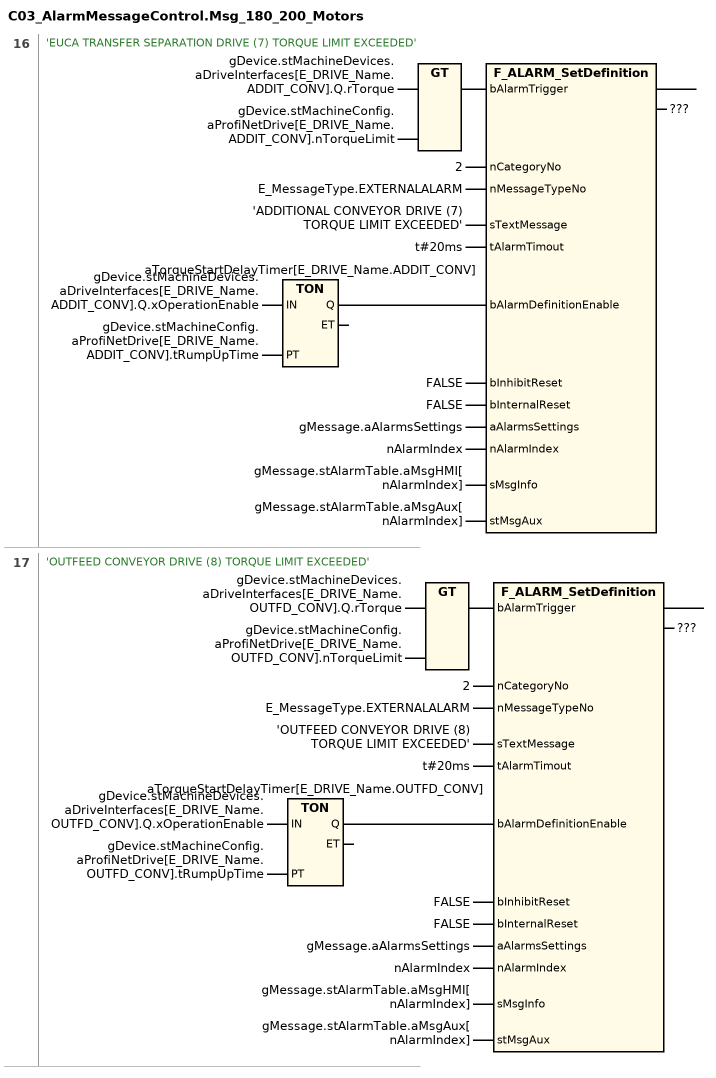
// NETWORK 16
// 'EUCA TRANSFER SEPARATION DRIVE (7) TORQUE LIMIT EXCEEDED'
aTorqueStartDelayTimer[E_DRIVE_Name.ADDIT_CONV](IN := gDevice.stMachineDevices.aDriveInterfaces[E_DRIVE_Name.ADDIT_CONV].Q.xOperationEnable, PT := gDevice.stMachineConfig.aProfiNetDrive[E_DRIVE_Name.ADDIT_CONV].tRumpUpTime); // TON
F_ALARM_SetDefinition(bAlarmTrigger := gDevice.stMachineDevices.aDriveInterfaces[E_DRIVE_Name.ADDIT_CONV].Q.rTorque > gDevice.stMachineConfig.aProfiNetDrive[E_DRIVE_Name.ADDIT_CONV].nTorqueLimit, nCategoryNo := 2, nMessageTypeNo := E_MessageType.EXTERNALALARM, sTextMessage := 'ADDITIONAL CONVEYOR DRIVE (7) TORQUE LIMIT EXCEEDED', tAlarmTimout := t#20ms, bAlarmDefinitionEnable := aTorqueStartDelayTimer[E_DRIVE_Name.ADDIT_CONV].Q, bInhibitReset := FALSE, bInternalReset := FALSE, aAlarmsSettings := gMessage.aAlarmsSettings, nAlarmIndex := nAlarmIndex, sMsgInfo := gMessage.stAlarmTable.aMsgHMI[nAlarmIndex], stMsgAux := gMessage.stAlarmTable.aMsgAux[nAlarmIndex]);

// NETWORK 17
// 'OUTFEED CONVEYOR DRIVE (8) TORQUE LIMIT EXCEEDED'
aTorqueStartDelayTimer[E_DRIVE_Name.OUTFD_CONV](IN := gDevice.stMachineDevices.aDriveInterfaces[E_DRIVE_Name.OUTFD_CONV].Q.xOperationEnable, PT := gDevice.stMachineConfig.aProfiNetDrive[E_DRIVE_Name.OUTFD_CONV].tRumpUpTime); // TON
F_ALARM_SetDefinition(bAlarmTrigger := gDevice.stMachineDevices.aDriveInterfaces[E_DRIVE_Name.OUTFD_CONV].Q.rTorque > gDevice.stMachineConfig.aProfiNetDrive[E_DRIVE_Name.OUTFD_CONV].nTorqueLimit, nCategoryNo := 2, nMessageTypeNo := E_MessageType.EXTERNALALARM, sTextMessage := 'OUTFEED CONVEYOR DRIVE (8) TORQUE LIMIT EXCEEDED', tAlarmTimout := t#20ms, bAlarmDefinitionEnable := aTorqueStartDelayTimer[E_DRIVE_Name.OUTFD_CONV].Q, bInhibitReset := FALSE, bInternalReset := FALSE, aAlarmsSettings := gMessage.aAlarmsSettings, nAlarmIndex := nAlarmIndex, sMsgInfo := gMessage.stAlarmTable.aMsgHMI[nAlarmIndex], stMsgAux := gMessage.stAlarmTable.aMsgAux[nAlarmIndex]);

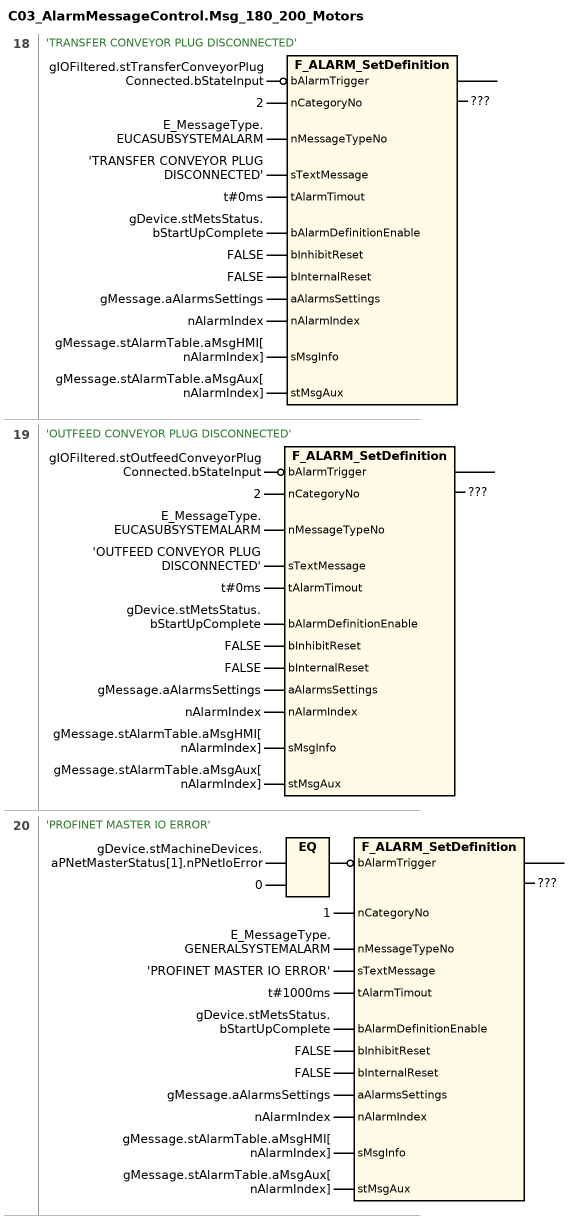
// NETWORK 18
// 'TRANSFER CONVEYOR PLUG DISCONNECTED'
F_ALARM_SetDefinition(bAlarmTrigger := NOT gIOFiltered.stTransferConveyorPlugConnected.bStateInput, nCategoryNo := 2, nMessageTypeNo := E_MessageType.EUCASUBSYSTEMALARM, sTextMessage := 'TRANSFER CONVEYOR PLUG DISCONNECTED', tAlarmTimout := t#0ms, bAlarmDefinitionEnable := gDevice.stMetsStatus.bStartUpComplete, bInhibitReset := FALSE, bInternalReset := FALSE, aAlarmsSettings := gMessage.aAlarmsSettings, nAlarmIndex := nAlarmIndex, sMsgInfo := gMessage.stAlarmTable.aMsgHMI[nAlarmIndex], stMsgAux := gMessage.stAlarmTable.aMsgAux[nAlarmIndex]);

// NETWORK 19
// 'OUTFEED CONVEYOR PLUG DISCONNECTED'
F_ALARM_SetDefinition(bAlarmTrigger := NOT gIOFiltered.stOutfeedConveyorPlugConnected.bStateInput, nCategoryNo := 2, nMessageTypeNo := E_MessageType.EUCASUBSYSTEMALARM, sTextMessage := 'OUTFEED CONVEYOR PLUG DISCONNECTED', tAlarmTimout := t#0ms, bAlarmDefinitionEnable := gDevice.stMetsStatus.bStartUpComplete, bInhibitReset := FALSE, bInternalReset := FALSE, aAlarmsSettings := gMessage.aAlarmsSettings, nAlarmIndex := nAlarmIndex, sMsgInfo := gMessage.stAlarmTable.aMsgHMI[nAlarmIndex], stMsgAux := gMessage.stAlarmTable.aMsgAux[nAlarmIndex]);

// NETWORK 20
// 'PROFINET MASTER IO ERROR'
F_ALARM_SetDefinition(bAlarmTrigger := NOT (gDevice.stMachineDevices.aPNetMasterStatus[1].nPNetIoError = 0), nCategoryNo := 1, nMessageTypeNo := E_MessageType.GENERALSYSTEMALARM, sTextMessage := 'PROFINET MASTER IO ERROR', tAlarmTimout := t#1000ms, bAlarmDefinitionEnable := gDevice.stMetsStatus.bStartUpComplete, bInhibitReset := FALSE, bInternalReset := FALSE, aAlarmsSettings := gMessage.aAlarmsSettings, nAlarmIndex := nAlarmIndex, sMsgInfo := gMessage.stAlarmTable.aMsgHMI[nAlarmIndex], stMsgAux := gMessage.stAlarmTable.aMsgAux[nAlarmIndex]);

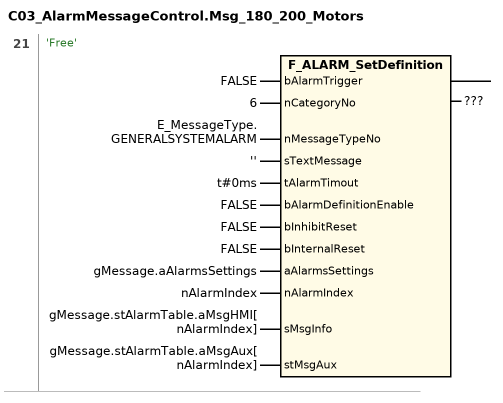
// NETWORK 21
// 'Free'
F_ALARM_SetDefinition(bAlarmTrigger := FALSE, nCategoryNo := 6, nMessageTypeNo := E_MessageType.GENERALSYSTEMALARM, sTextMessage := '', tAlarmTimout := t#0ms, bAlarmDefinitionEnable := FALSE, bInhibitReset := FALSE, bInternalReset := FALSE, aAlarmsSettings := gMessage.aAlarmsSettings, nAlarmIndex := nAlarmIndex, sMsgInfo := gMessage.stAlarmTable.aMsgHMI[nAlarmIndex], stMsgAux := gMessage.stAlarmTable.aMsgAux[nAlarmIndex]);
END_ACTION

ACTION Msg_201_208_Interface:
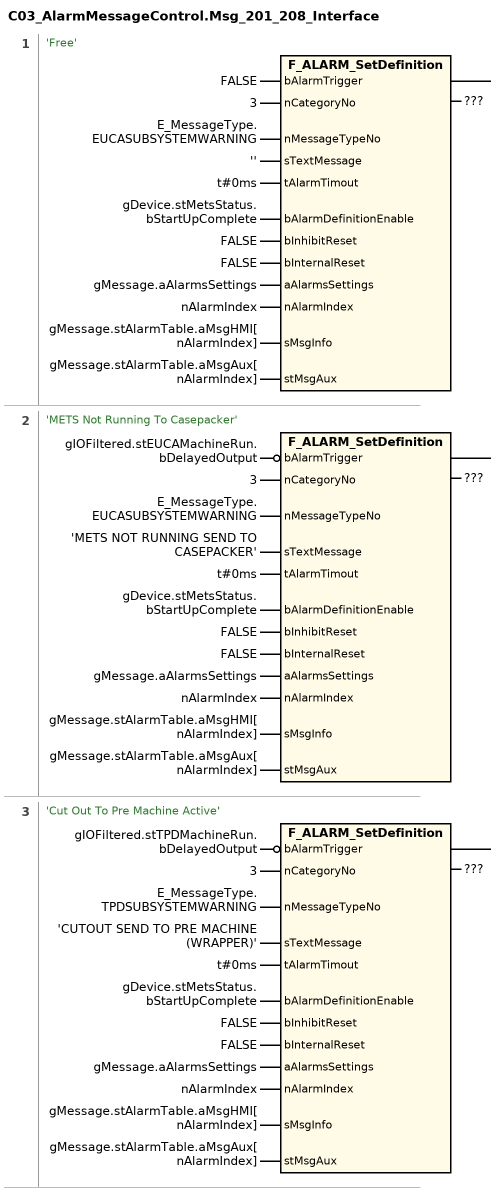
// NETWORK 1
// 'Free'
F_ALARM_SetDefinition(bAlarmTrigger := FALSE, nCategoryNo := 3, nMessageTypeNo := E_MessageType.EUCASUBSYSTEMWARNING, sTextMessage := '', tAlarmTimout := t#0ms, bAlarmDefinitionEnable := gDevice.stMetsStatus.bStartUpComplete, bInhibitReset := FALSE, bInternalReset := FALSE, aAlarmsSettings := gMessage.aAlarmsSettings, nAlarmIndex := nAlarmIndex, sMsgInfo := gMessage.stAlarmTable.aMsgHMI[nAlarmIndex], stMsgAux := gMessage.stAlarmTable.aMsgAux[nAlarmIndex]);

// NETWORK 2
// 'METS Not Running To Casepacker'
F_ALARM_SetDefinition(bAlarmTrigger := NOT gIOFiltered.stEUCAMachineRun.bDelayedOutput, nCategoryNo := 3, nMessageTypeNo := E_MessageType.EUCASUBSYSTEMWARNING, sTextMessage := 'METS NOT RUNNING SEND TO CASEPACKER', tAlarmTimout := t#0ms, bAlarmDefinitionEnable := gDevice.stMetsStatus.bStartUpComplete, bInhibitReset := FALSE, bInternalReset := FALSE, aAlarmsSettings := gMessage.aAlarmsSettings, nAlarmIndex := nAlarmIndex, sMsgInfo := gMessage.stAlarmTable.aMsgHMI[nAlarmIndex], stMsgAux := gMessage.stAlarmTable.aMsgAux[nAlarmIndex]);

// NETWORK 3
// 'Cut Out To Pre Machine Active'
F_ALARM_SetDefinition(bAlarmTrigger := NOT gIOFiltered.stTPDMachineRun.bDelayedOutput, nCategoryNo := 3, nMessageTypeNo := E_MessageType.TPDSUBSYSTEMWARNING, sTextMessage := 'CUTOUT SEND TO PRE MACHINE (WRAPPER)', tAlarmTimout := t#0ms, bAlarmDefinitionEnable := gDevice.stMetsStatus.bStartUpComplete, bInhibitReset := FALSE, bInternalReset := FALSE, aAlarmsSettings := gMessage.aAlarmsSettings, nAlarmIndex := nAlarmIndex, sMsgInfo := gMessage.stAlarmTable.aMsgHMI[nAlarmIndex], stMsgAux := gMessage.stAlarmTable.aMsgAux[nAlarmIndex]);

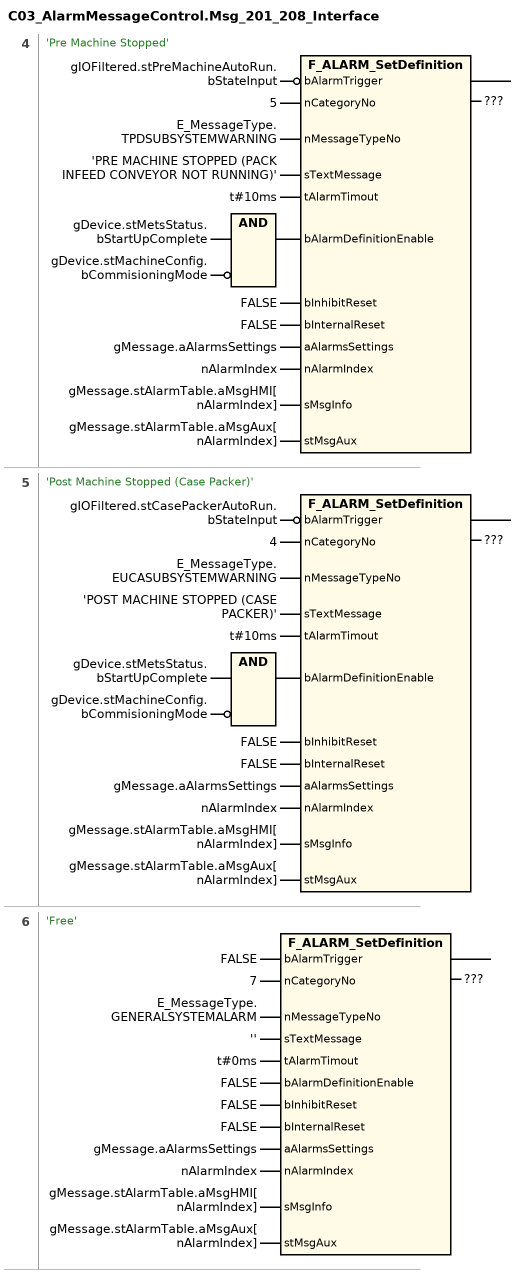
// NETWORK 4
// 'Pre Machine Stopped'
F_ALARM_SetDefinition(bAlarmTrigger := NOT gIOFiltered.stPreMachineAutoRun.bStateInput, nCategoryNo := 5, nMessageTypeNo := E_MessageType.TPDSUBSYSTEMWARNING, sTextMessage := 'PRE MACHINE STOPPED (PACK INFEED CONVEYOR NOT RUNNING)', tAlarmTimout := t#10ms, bAlarmDefinitionEnable := gDevice.stMetsStatus.bStartUpComplete AND NOT gDevice.stMachineConfig.bCommisioningMode, bInhibitReset := FALSE, bInternalReset := FALSE, aAlarmsSettings := gMessage.aAlarmsSettings, nAlarmIndex := nAlarmIndex, sMsgInfo := gMessage.stAlarmTable.aMsgHMI[nAlarmIndex], stMsgAux := gMessage.stAlarmTable.aMsgAux[nAlarmIndex]);

// NETWORK 5
// 'Post Machine Stopped (Case Packer)'
F_ALARM_SetDefinition(bAlarmTrigger := NOT gIOFiltered.stCasePackerAutoRun.bStateInput, nCategoryNo := 4, nMessageTypeNo := E_MessageType.EUCASUBSYSTEMWARNING, sTextMessage := 'POST MACHINE STOPPED (CASE PACKER)', tAlarmTimout := t#10ms, bAlarmDefinitionEnable := gDevice.stMetsStatus.bStartUpComplete AND NOT gDevice.stMachineConfig.bCommisioningMode, bInhibitReset := FALSE, bInternalReset := FALSE, aAlarmsSettings := gMessage.aAlarmsSettings, nAlarmIndex := nAlarmIndex, sMsgInfo := gMessage.stAlarmTable.aMsgHMI[nAlarmIndex], stMsgAux := gMessage.stAlarmTable.aMsgAux[nAlarmIndex]);

// NETWORK 6
// 'Free'
F_ALARM_SetDefinition(bAlarmTrigger := FALSE, nCategoryNo := 7, nMessageTypeNo := E_MessageType.GENERALSYSTEMALARM, sTextMessage := '', tAlarmTimout := t#0ms, bAlarmDefinitionEnable := FALSE, bInhibitReset := FALSE, bInternalReset := FALSE, aAlarmsSettings := gMessage.aAlarmsSettings, nAlarmIndex := nAlarmIndex, sMsgInfo := gMessage.stAlarmTable.aMsgHMI[nAlarmIndex], stMsgAux := gMessage.stAlarmTable.aMsgAux[nAlarmIndex]);

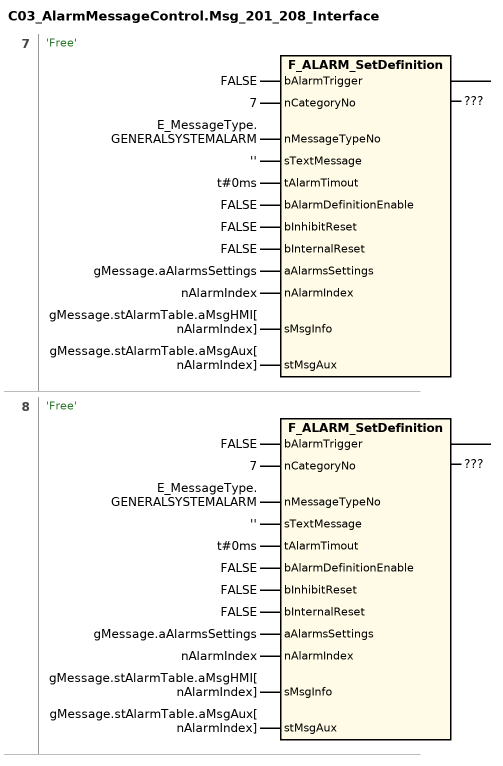
// NETWORK 7
// 'Free'
F_ALARM_SetDefinition(bAlarmTrigger := FALSE, nCategoryNo := 7, nMessageTypeNo := E_MessageType.GENERALSYSTEMALARM, sTextMessage := '', tAlarmTimout := t#0ms, bAlarmDefinitionEnable := FALSE, bInhibitReset := FALSE, bInternalReset := FALSE, aAlarmsSettings := gMessage.aAlarmsSettings, nAlarmIndex := nAlarmIndex, sMsgInfo := gMessage.stAlarmTable.aMsgHMI[nAlarmIndex], stMsgAux := gMessage.stAlarmTable.aMsgAux[nAlarmIndex]);

// NETWORK 8
// 'Free'
F_ALARM_SetDefinition(bAlarmTrigger := FALSE, nCategoryNo := 7, nMessageTypeNo := E_MessageType.GENERALSYSTEMALARM, sTextMessage := '', tAlarmTimout := t#0ms, bAlarmDefinitionEnable := FALSE, bInhibitReset := FALSE, bInternalReset := FALSE, aAlarmsSettings := gMessage.aAlarmsSettings, nAlarmIndex := nAlarmIndex, sMsgInfo := gMessage.stAlarmTable.aMsgHMI[nAlarmIndex], stMsgAux := gMessage.stAlarmTable.aMsgAux[nAlarmIndex]);
END_ACTION

ACTION Msg_209_237_Labellers:
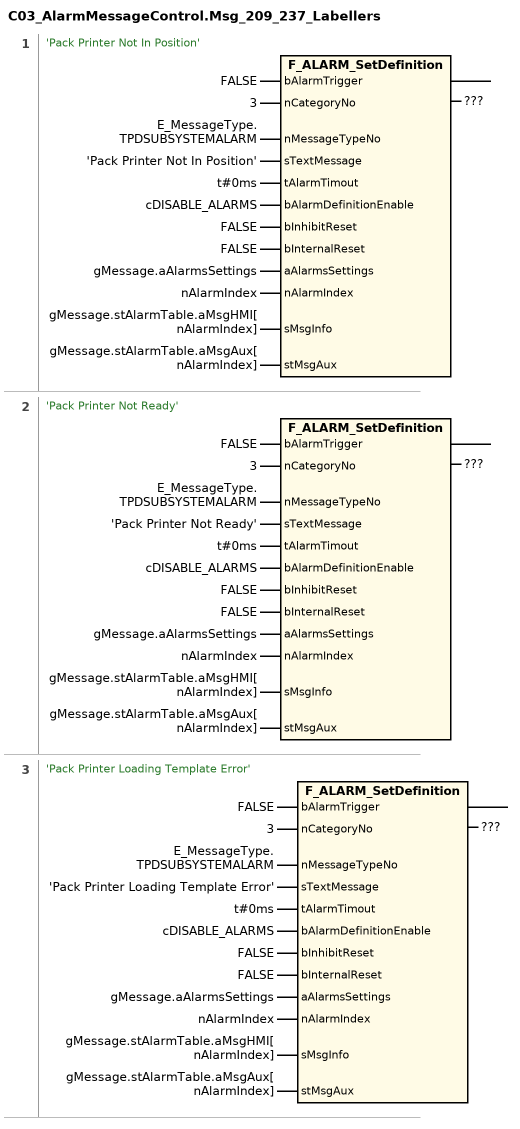
// NETWORK 1
// 'Pack Printer Not In Position'
F_ALARM_SetDefinition(bAlarmTrigger := FALSE, nCategoryNo := 3, nMessageTypeNo := E_MessageType.TPDSUBSYSTEMALARM, sTextMessage := 'Pack Printer Not In Position', tAlarmTimout := t#0ms, bAlarmDefinitionEnable := cDISABLE_ALARMS, bInhibitReset := FALSE, bInternalReset := FALSE, aAlarmsSettings := gMessage.aAlarmsSettings, nAlarmIndex := nAlarmIndex, sMsgInfo := gMessage.stAlarmTable.aMsgHMI[nAlarmIndex], stMsgAux := gMessage.stAlarmTable.aMsgAux[nAlarmIndex]);

// NETWORK 2
// 'Pack Printer Not Ready'
F_ALARM_SetDefinition(bAlarmTrigger := FALSE, nCategoryNo := 3, nMessageTypeNo := E_MessageType.TPDSUBSYSTEMALARM, sTextMessage := 'Pack Printer Not Ready', tAlarmTimout := t#0ms, bAlarmDefinitionEnable := cDISABLE_ALARMS, bInhibitReset := FALSE, bInternalReset := FALSE, aAlarmsSettings := gMessage.aAlarmsSettings, nAlarmIndex := nAlarmIndex, sMsgInfo := gMessage.stAlarmTable.aMsgHMI[nAlarmIndex], stMsgAux := gMessage.stAlarmTable.aMsgAux[nAlarmIndex]);

// NETWORK 3
// 'Pack Printer Loading Template Error'
F_ALARM_SetDefinition(bAlarmTrigger := FALSE, nCategoryNo := 3, nMessageTypeNo := E_MessageType.TPDSUBSYSTEMALARM, sTextMessage := 'Pack Printer Loading Template Error', tAlarmTimout := t#0ms, bAlarmDefinitionEnable := cDISABLE_ALARMS, bInhibitReset := FALSE, bInternalReset := FALSE, aAlarmsSettings := gMessage.aAlarmsSettings, nAlarmIndex := nAlarmIndex, sMsgInfo := gMessage.stAlarmTable.aMsgHMI[nAlarmIndex], stMsgAux := gMessage.stAlarmTable.aMsgAux[nAlarmIndex]);

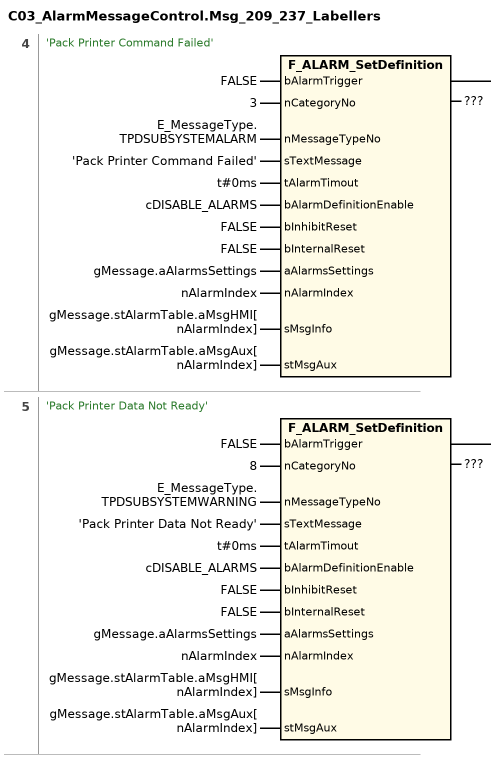
// NETWORK 4
// 'Pack Printer Command Failed'
F_ALARM_SetDefinition(bAlarmTrigger := FALSE, nCategoryNo := 3, nMessageTypeNo := E_MessageType.TPDSUBSYSTEMALARM, sTextMessage := 'Pack Printer Command Failed', tAlarmTimout := t#0ms, bAlarmDefinitionEnable := cDISABLE_ALARMS, bInhibitReset := FALSE, bInternalReset := FALSE, aAlarmsSettings := gMessage.aAlarmsSettings, nAlarmIndex := nAlarmIndex, sMsgInfo := gMessage.stAlarmTable.aMsgHMI[nAlarmIndex], stMsgAux := gMessage.stAlarmTable.aMsgAux[nAlarmIndex]);

// NETWORK 5
// 'Pack Printer Data Not Ready'
F_ALARM_SetDefinition(bAlarmTrigger := FALSE, nCategoryNo := 8, nMessageTypeNo := E_MessageType.TPDSUBSYSTEMWARNING, sTextMessage := 'Pack Printer Data Not Ready', tAlarmTimout := t#0ms, bAlarmDefinitionEnable := cDISABLE_ALARMS, bInhibitReset := FALSE, bInternalReset := FALSE, aAlarmsSettings := gMessage.aAlarmsSettings, nAlarmIndex := nAlarmIndex, sMsgInfo := gMessage.stAlarmTable.aMsgHMI[nAlarmIndex], stMsgAux := gMessage.stAlarmTable.aMsgAux[nAlarmIndex]);

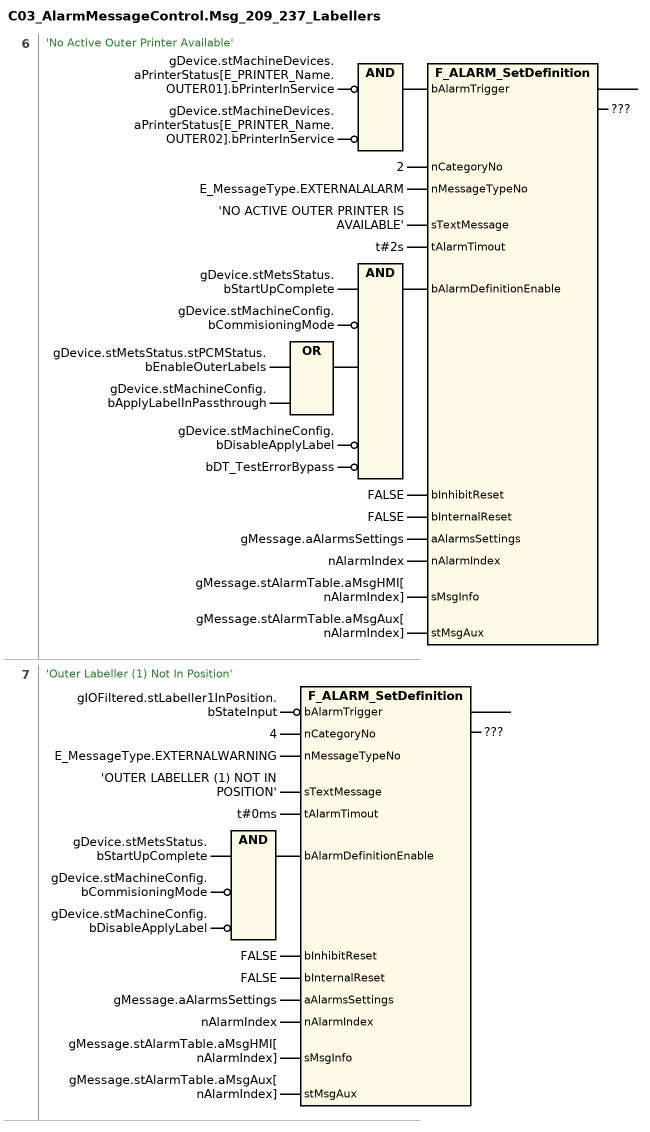
// NETWORK 6
// 'No Active Outer Printer Available'
F_ALARM_SetDefinition(bAlarmTrigger := NOT gDevice.stMachineDevices.aPrinterStatus[E_PRINTER_Name.OUTER01].bPrinterInService AND NOT gDevice.stMachineDevices.aPrinterStatus[E_PRINTER_Name.OUTER02].bPrinterInService, nCategoryNo := 2, nMessageTypeNo := E_MessageType.EXTERNALALARM, sTextMessage := 'NO ACTIVE OUTER PRINTER IS AVAILABLE', tAlarmTimout := t#2s, bAlarmDefinitionEnable := gDevice.stMetsStatus.bStartUpComplete AND NOT gDevice.stMachineConfig.bCommisioningMode AND (gDevice.stMetsStatus.stPCMStatus.bEnableOuterLabels OR gDevice.stMachineConfig.bApplyLabelInPassthrough) AND NOT gDevice.stMachineConfig.bDisableApplyLabel AND NOT bDT_TestErrorBypass, bInhibitReset := FALSE, bInternalReset := FALSE, aAlarmsSettings := gMessage.aAlarmsSettings, nAlarmIndex := nAlarmIndex, sMsgInfo := gMessage.stAlarmTable.aMsgHMI[nAlarmIndex], stMsgAux := gMessage.stAlarmTable.aMsgAux[nAlarmIndex]);

// NETWORK 7
// 'Outer Labeller (1) Not In Position'
F_ALARM_SetDefinition(bAlarmTrigger := NOT gIOFiltered.stLabeller1InPosition.bStateInput, nCategoryNo := 4, nMessageTypeNo := E_MessageType.EXTERNALWARNING, sTextMessage := 'OUTER LABELLER (1) NOT IN POSITION', tAlarmTimout := t#0ms, bAlarmDefinitionEnable := gDevice.stMetsStatus.bStartUpComplete AND NOT gDevice.stMachineConfig.bCommisioningMode AND NOT gDevice.stMachineConfig.bDisableApplyLabel, bInhibitReset := FALSE, bInternalReset := FALSE, aAlarmsSettings := gMessage.aAlarmsSettings, nAlarmIndex := nAlarmIndex, sMsgInfo := gMessage.stAlarmTable.aMsgHMI[nAlarmIndex], stMsgAux := gMessage.stAlarmTable.aMsgAux[nAlarmIndex]);

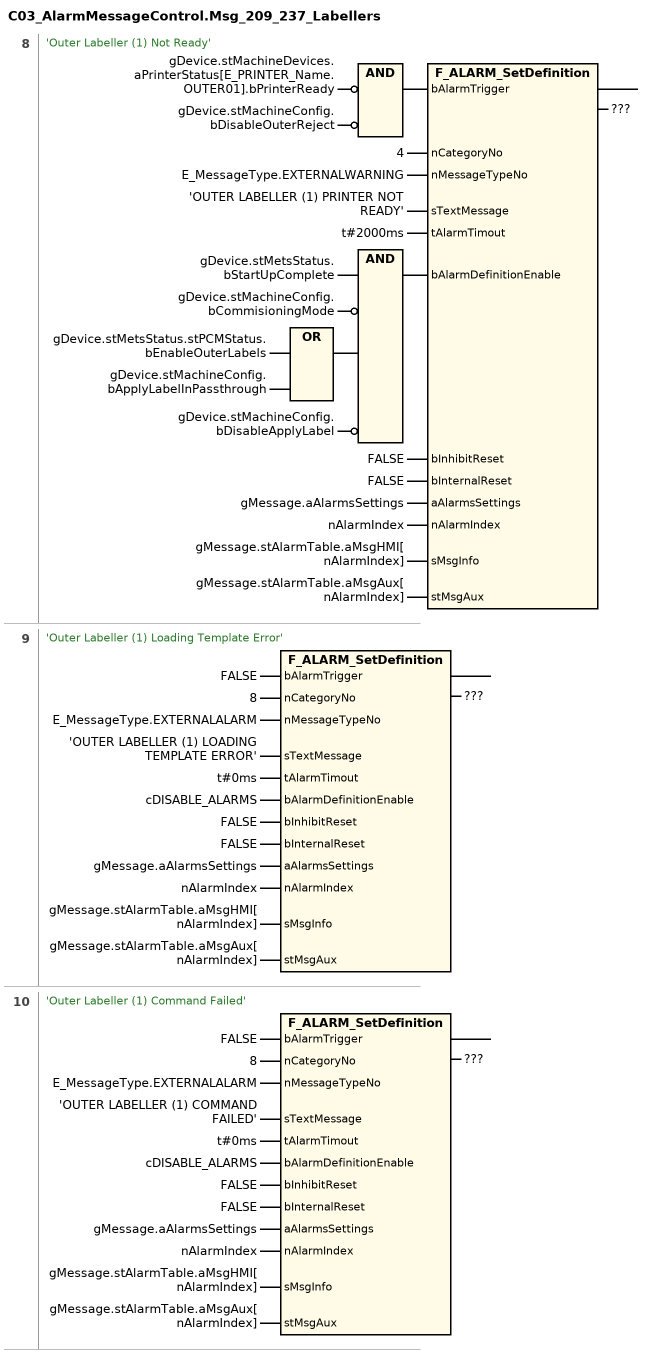
// NETWORK 8
// 'Outer Labeller (1) Not Ready'
F_ALARM_SetDefinition(bAlarmTrigger := NOT gDevice.stMachineDevices.aPrinterStatus[E_PRINTER_Name.OUTER01].bPrinterReady AND NOT gDevice.stMachineConfig.bDisableOuterReject, nCategoryNo := 4, nMessageTypeNo := E_MessageType.EXTERNALWARNING, sTextMessage := 'OUTER LABELLER (1) PRINTER NOT READY', tAlarmTimout := t#2000ms, bAlarmDefinitionEnable := gDevice.stMetsStatus.bStartUpComplete AND NOT gDevice.stMachineConfig.bCommisioningMode AND (gDevice.stMetsStatus.stPCMStatus.bEnableOuterLabels OR gDevice.stMachineConfig.bApplyLabelInPassthrough) AND NOT gDevice.stMachineConfig.bDisableApplyLabel, bInhibitReset := FALSE, bInternalReset := FALSE, aAlarmsSettings := gMessage.aAlarmsSettings, nAlarmIndex := nAlarmIndex, sMsgInfo := gMessage.stAlarmTable.aMsgHMI[nAlarmIndex], stMsgAux := gMessage.stAlarmTable.aMsgAux[nAlarmIndex]);

// NETWORK 9
// 'Outer Labeller (1) Loading Template Error'
F_ALARM_SetDefinition(bAlarmTrigger := FALSE, nCategoryNo := 8, nMessageTypeNo := E_MessageType.EXTERNALALARM, sTextMessage := 'OUTER LABELLER (1) LOADING TEMPLATE ERROR', tAlarmTimout := t#0ms, bAlarmDefinitionEnable := cDISABLE_ALARMS, bInhibitReset := FALSE, bInternalReset := FALSE, aAlarmsSettings := gMessage.aAlarmsSettings, nAlarmIndex := nAlarmIndex, sMsgInfo := gMessage.stAlarmTable.aMsgHMI[nAlarmIndex], stMsgAux := gMessage.stAlarmTable.aMsgAux[nAlarmIndex]);

// NETWORK 10
// 'Outer Labeller (1) Command Failed'
F_ALARM_SetDefinition(bAlarmTrigger := FALSE, nCategoryNo := 8, nMessageTypeNo := E_MessageType.EXTERNALALARM, sTextMessage := 'OUTER LABELLER (1) COMMAND FAILED', tAlarmTimout := t#0ms, bAlarmDefinitionEnable := cDISABLE_ALARMS, bInhibitReset := FALSE, bInternalReset := FALSE, aAlarmsSettings := gMessage.aAlarmsSettings, nAlarmIndex := nAlarmIndex, sMsgInfo := gMessage.stAlarmTable.aMsgHMI[nAlarmIndex], stMsgAux := gMessage.stAlarmTable.aMsgAux[nAlarmIndex]);

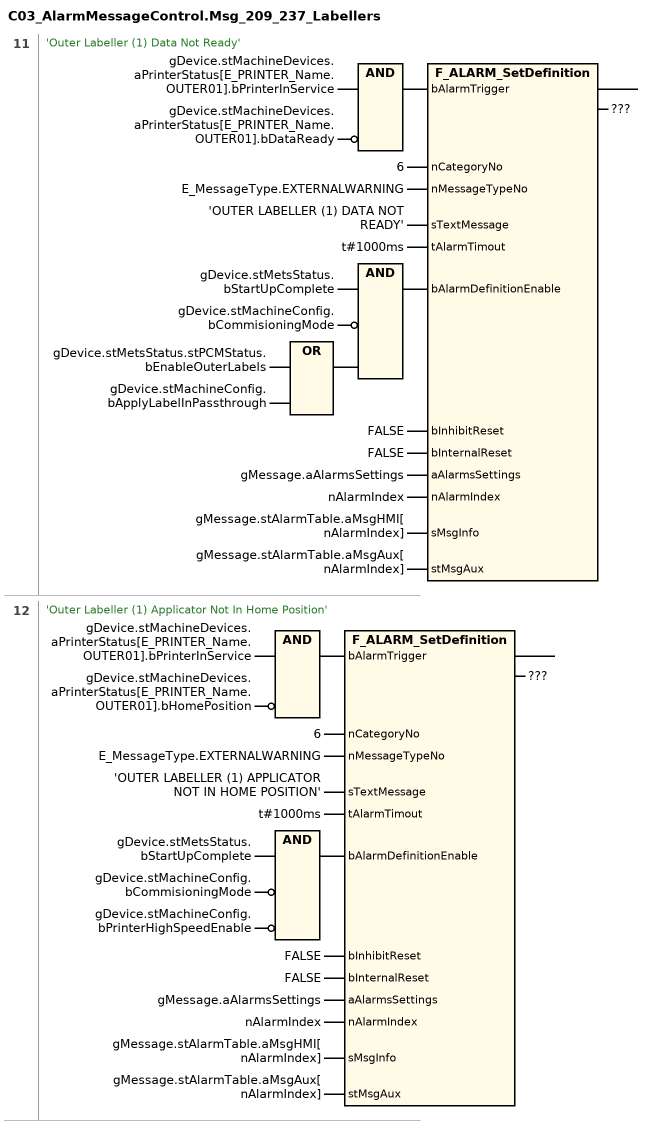
// NETWORK 11
// 'Outer Labeller (1) Data Not Ready'
F_ALARM_SetDefinition(bAlarmTrigger := gDevice.stMachineDevices.aPrinterStatus[E_PRINTER_Name.OUTER01].bPrinterInService AND NOT gDevice.stMachineDevices.aPrinterStatus[E_PRINTER_Name.OUTER01].bDataReady, nCategoryNo := 6, nMessageTypeNo := E_MessageType.EXTERNALWARNING, sTextMessage := 'OUTER LABELLER (1) DATA NOT READY', tAlarmTimout := t#1000ms, bAlarmDefinitionEnable := gDevice.stMetsStatus.bStartUpComplete AND NOT gDevice.stMachineConfig.bCommisioningMode AND (gDevice.stMetsStatus.stPCMStatus.bEnableOuterLabels OR gDevice.stMachineConfig.bApplyLabelInPassthrough), bInhibitReset := FALSE, bInternalReset := FALSE, aAlarmsSettings := gMessage.aAlarmsSettings, nAlarmIndex := nAlarmIndex, sMsgInfo := gMessage.stAlarmTable.aMsgHMI[nAlarmIndex], stMsgAux := gMessage.stAlarmTable.aMsgAux[nAlarmIndex]);

// NETWORK 12
// 'Outer Labeller (1) Applicator Not In Home Position'
F_ALARM_SetDefinition(bAlarmTrigger := gDevice.stMachineDevices.aPrinterStatus[E_PRINTER_Name.OUTER01].bPrinterInService AND NOT gDevice.stMachineDevices.aPrinterStatus[E_PRINTER_Name.OUTER01].bHomePosition, nCategoryNo := 6, nMessageTypeNo := E_MessageType.EXTERNALWARNING, sTextMessage := 'OUTER LABELLER (1) APPLICATOR NOT IN HOME POSITION', tAlarmTimout := t#1000ms, bAlarmDefinitionEnable := gDevice.stMetsStatus.bStartUpComplete AND NOT gDevice.stMachineConfig.bCommisioningMode AND NOT gDevice.stMachineConfig.bPrinterHighSpeedEnable, bInhibitReset := FALSE, bInternalReset := FALSE, aAlarmsSettings := gMessage.aAlarmsSettings, nAlarmIndex := nAlarmIndex, sMsgInfo := gMessage.stAlarmTable.aMsgHMI[nAlarmIndex], stMsgAux := gMessage.stAlarmTable.aMsgAux[nAlarmIndex]);

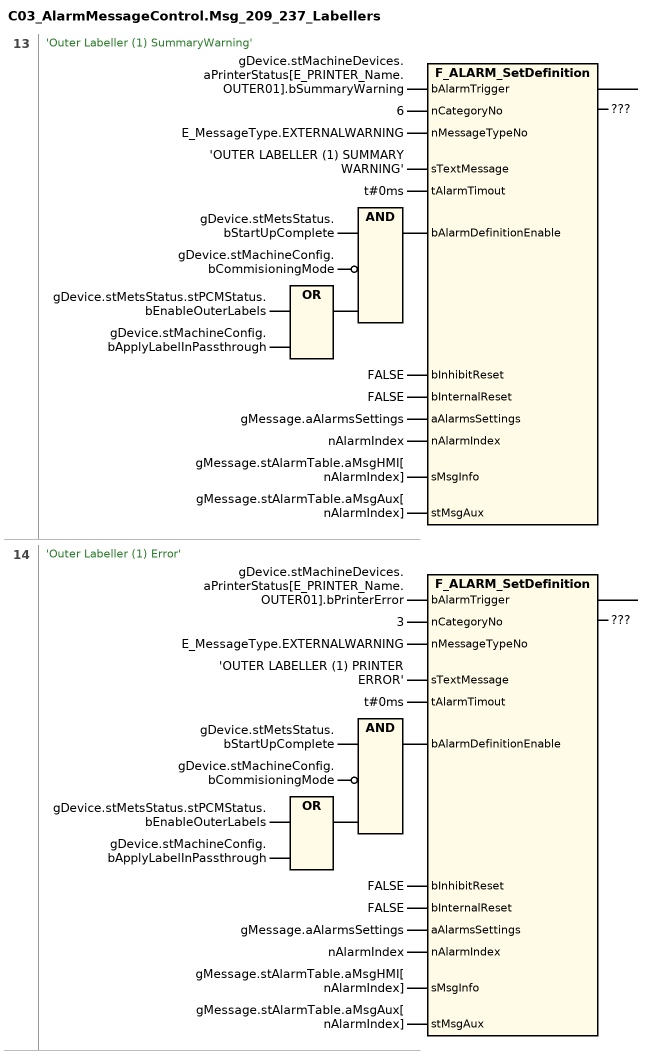
// NETWORK 13
// 'Outer Labeller (1) SummaryWarning'
F_ALARM_SetDefinition(bAlarmTrigger := gDevice.stMachineDevices.aPrinterStatus[E_PRINTER_Name.OUTER01].bSummaryWarning, nCategoryNo := 6, nMessageTypeNo := E_MessageType.EXTERNALWARNING, sTextMessage := 'OUTER LABELLER (1) SUMMARY WARNING', tAlarmTimout := t#0ms, bAlarmDefinitionEnable := gDevice.stMetsStatus.bStartUpComplete AND NOT gDevice.stMachineConfig.bCommisioningMode AND (gDevice.stMetsStatus.stPCMStatus.bEnableOuterLabels OR gDevice.stMachineConfig.bApplyLabelInPassthrough), bInhibitReset := FALSE, bInternalReset := FALSE, aAlarmsSettings := gMessage.aAlarmsSettings, nAlarmIndex := nAlarmIndex, sMsgInfo := gMessage.stAlarmTable.aMsgHMI[nAlarmIndex], stMsgAux := gMessage.stAlarmTable.aMsgAux[nAlarmIndex]);

// NETWORK 14
// 'Outer Labeller (1) Error'
F_ALARM_SetDefinition(bAlarmTrigger := gDevice.stMachineDevices.aPrinterStatus[E_PRINTER_Name.OUTER01].bPrinterError, nCategoryNo := 3, nMessageTypeNo := E_MessageType.EXTERNALWARNING, sTextMessage := 'OUTER LABELLER (1) PRINTER ERROR', tAlarmTimout := t#0ms, bAlarmDefinitionEnable := gDevice.stMetsStatus.bStartUpComplete AND NOT gDevice.stMachineConfig.bCommisioningMode AND (gDevice.stMetsStatus.stPCMStatus.bEnableOuterLabels OR gDevice.stMachineConfig.bApplyLabelInPassthrough), bInhibitReset := FALSE, bInternalReset := FALSE, aAlarmsSettings := gMessage.aAlarmsSettings, nAlarmIndex := nAlarmIndex, sMsgInfo := gMessage.stAlarmTable.aMsgHMI[nAlarmIndex], stMsgAux := gMessage.stAlarmTable.aMsgAux[nAlarmIndex]);

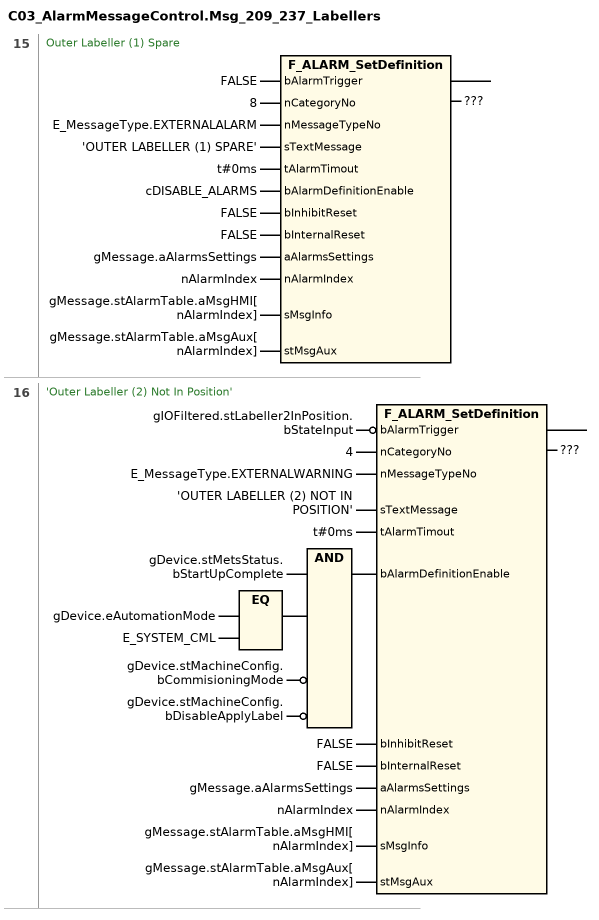
// NETWORK 15
// Outer Labeller (1) Spare
F_ALARM_SetDefinition(bAlarmTrigger := FALSE, nCategoryNo := 8, nMessageTypeNo := E_MessageType.EXTERNALALARM, sTextMessage := 'OUTER LABELLER (1) SPARE', tAlarmTimout := t#0ms, bAlarmDefinitionEnable := cDISABLE_ALARMS, bInhibitReset := FALSE, bInternalReset := FALSE, aAlarmsSettings := gMessage.aAlarmsSettings, nAlarmIndex := nAlarmIndex, sMsgInfo := gMessage.stAlarmTable.aMsgHMI[nAlarmIndex], stMsgAux := gMessage.stAlarmTable.aMsgAux[nAlarmIndex]);

// NETWORK 16
// 'Outer Labeller (2) Not In Position'
F_ALARM_SetDefinition(bAlarmTrigger := NOT gIOFiltered.stLabeller2InPosition.bStateInput, nCategoryNo := 4, nMessageTypeNo := E_MessageType.EXTERNALWARNING, sTextMessage := 'OUTER LABELLER (2) NOT IN POSITION', tAlarmTimout := t#0ms, bAlarmDefinitionEnable := gDevice.stMetsStatus.bStartUpComplete AND gDevice.eAutomationMode = E_SYSTEM_CML AND NOT gDevice.stMachineConfig.bCommisioningMode AND NOT gDevice.stMachineConfig.bDisableApplyLabel, bInhibitReset := FALSE, bInternalReset := FALSE, aAlarmsSettings := gMessage.aAlarmsSettings, nAlarmIndex := nAlarmIndex, sMsgInfo := gMessage.stAlarmTable.aMsgHMI[nAlarmIndex], stMsgAux := gMessage.stAlarmTable.aMsgAux[nAlarmIndex]);

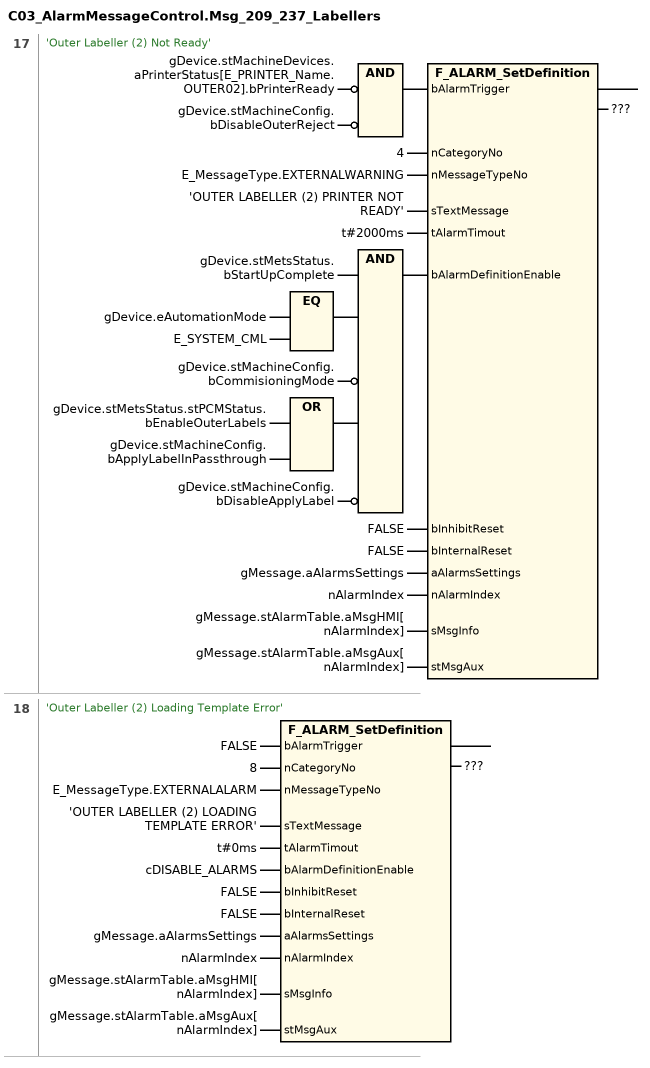
// NETWORK 17
// 'Outer Labeller (2) Not Ready'
F_ALARM_SetDefinition(bAlarmTrigger := NOT gDevice.stMachineDevices.aPrinterStatus[E_PRINTER_Name.OUTER02].bPrinterReady AND NOT gDevice.stMachineConfig.bDisableOuterReject, nCategoryNo := 4, nMessageTypeNo := E_MessageType.EXTERNALWARNING, sTextMessage := 'OUTER LABELLER (2) PRINTER NOT READY', tAlarmTimout := t#2000ms, bAlarmDefinitionEnable := gDevice.stMetsStatus.bStartUpComplete AND gDevice.eAutomationMode = E_SYSTEM_CML AND NOT gDevice.stMachineConfig.bCommisioningMode AND (gDevice.stMetsStatus.stPCMStatus.bEnableOuterLabels OR gDevice.stMachineConfig.bApplyLabelInPassthrough) AND NOT gDevice.stMachineConfig.bDisableApplyLabel, bInhibitReset := FALSE, bInternalReset := FALSE, aAlarmsSettings := gMessage.aAlarmsSettings, nAlarmIndex := nAlarmIndex, sMsgInfo := gMessage.stAlarmTable.aMsgHMI[nAlarmIndex], stMsgAux := gMessage.stAlarmTable.aMsgAux[nAlarmIndex]);

// NETWORK 18
// 'Outer Labeller (2) Loading Template Error'
F_ALARM_SetDefinition(bAlarmTrigger := FALSE, nCategoryNo := 8, nMessageTypeNo := E_MessageType.EXTERNALALARM, sTextMessage := 'OUTER LABELLER (2) LOADING TEMPLATE ERROR', tAlarmTimout := t#0ms, bAlarmDefinitionEnable := cDISABLE_ALARMS, bInhibitReset := FALSE, bInternalReset := FALSE, aAlarmsSettings := gMessage.aAlarmsSettings, nAlarmIndex := nAlarmIndex, sMsgInfo := gMessage.stAlarmTable.aMsgHMI[nAlarmIndex], stMsgAux := gMessage.stAlarmTable.aMsgAux[nAlarmIndex]);

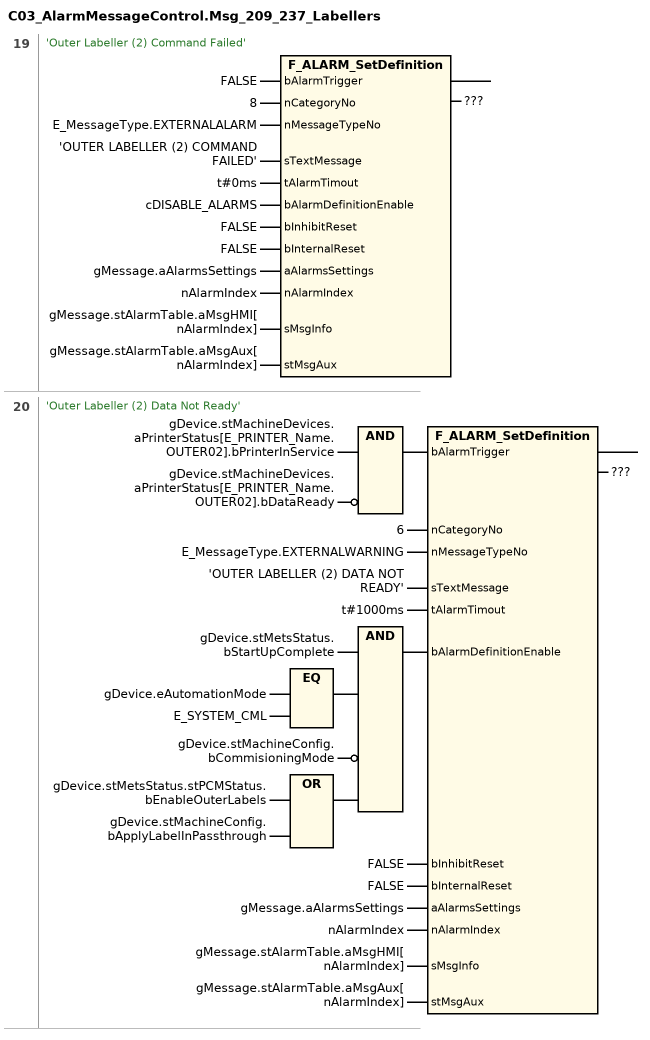
// NETWORK 19
// 'Outer Labeller (2) Command Failed'
F_ALARM_SetDefinition(bAlarmTrigger := FALSE, nCategoryNo := 8, nMessageTypeNo := E_MessageType.EXTERNALALARM, sTextMessage := 'OUTER LABELLER (2) COMMAND FAILED', tAlarmTimout := t#0ms, bAlarmDefinitionEnable := cDISABLE_ALARMS, bInhibitReset := FALSE, bInternalReset := FALSE, aAlarmsSettings := gMessage.aAlarmsSettings, nAlarmIndex := nAlarmIndex, sMsgInfo := gMessage.stAlarmTable.aMsgHMI[nAlarmIndex], stMsgAux := gMessage.stAlarmTable.aMsgAux[nAlarmIndex]);

// NETWORK 20
// 'Outer Labeller (2) Data Not Ready'
F_ALARM_SetDefinition(bAlarmTrigger := gDevice.stMachineDevices.aPrinterStatus[E_PRINTER_Name.OUTER02].bPrinterInService AND NOT gDevice.stMachineDevices.aPrinterStatus[E_PRINTER_Name.OUTER02].bDataReady, nCategoryNo := 6, nMessageTypeNo := E_MessageType.EXTERNALWARNING, sTextMessage := 'OUTER LABELLER (2) DATA NOT READY', tAlarmTimout := t#1000ms, bAlarmDefinitionEnable := gDevice.stMetsStatus.bStartUpComplete AND gDevice.eAutomationMode = E_SYSTEM_CML AND NOT gDevice.stMachineConfig.bCommisioningMode AND (gDevice.stMetsStatus.stPCMStatus.bEnableOuterLabels OR gDevice.stMachineConfig.bApplyLabelInPassthrough), bInhibitReset := FALSE, bInternalReset := FALSE, aAlarmsSettings := gMessage.aAlarmsSettings, nAlarmIndex := nAlarmIndex, sMsgInfo := gMessage.stAlarmTable.aMsgHMI[nAlarmIndex], stMsgAux := gMessage.stAlarmTable.aMsgAux[nAlarmIndex]);

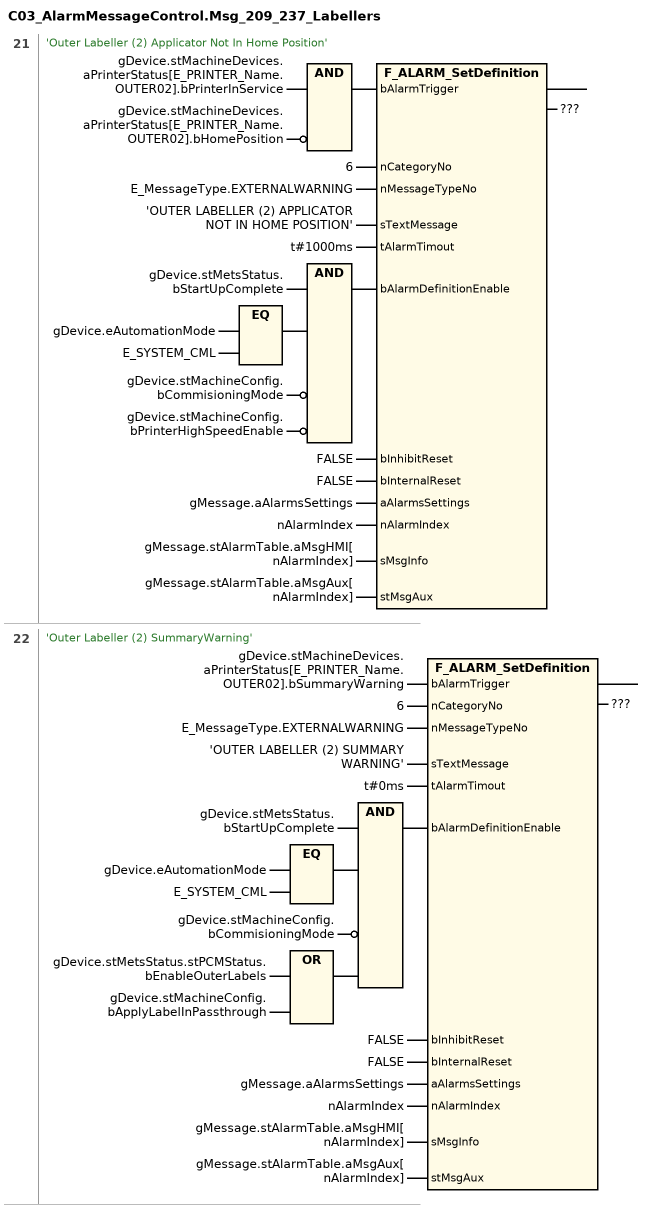
// NETWORK 21
// 'Outer Labeller (2) Applicator Not In Home Position'
F_ALARM_SetDefinition(bAlarmTrigger := gDevice.stMachineDevices.aPrinterStatus[E_PRINTER_Name.OUTER02].bPrinterInService AND NOT gDevice.stMachineDevices.aPrinterStatus[E_PRINTER_Name.OUTER02].bHomePosition, nCategoryNo := 6, nMessageTypeNo := E_MessageType.EXTERNALWARNING, sTextMessage := 'OUTER LABELLER (2) APPLICATOR NOT IN HOME POSITION', tAlarmTimout := t#1000ms, bAlarmDefinitionEnable := gDevice.stMetsStatus.bStartUpComplete AND gDevice.eAutomationMode = E_SYSTEM_CML AND NOT gDevice.stMachineConfig.bCommisioningMode AND NOT gDevice.stMachineConfig.bPrinterHighSpeedEnable, bInhibitReset := FALSE, bInternalReset := FALSE, aAlarmsSettings := gMessage.aAlarmsSettings, nAlarmIndex := nAlarmIndex, sMsgInfo := gMessage.stAlarmTable.aMsgHMI[nAlarmIndex], stMsgAux := gMessage.stAlarmTable.aMsgAux[nAlarmIndex]);

// NETWORK 22
// 'Outer Labeller (2) SummaryWarning'
F_ALARM_SetDefinition(bAlarmTrigger := gDevice.stMachineDevices.aPrinterStatus[E_PRINTER_Name.OUTER02].bSummaryWarning, nCategoryNo := 6, nMessageTypeNo := E_MessageType.EXTERNALWARNING, sTextMessage := 'OUTER LABELLER (2) SUMMARY WARNING', tAlarmTimout := t#0ms, bAlarmDefinitionEnable := gDevice.stMetsStatus.bStartUpComplete AND gDevice.eAutomationMode = E_SYSTEM_CML AND NOT gDevice.stMachineConfig.bCommisioningMode AND (gDevice.stMetsStatus.stPCMStatus.bEnableOuterLabels OR gDevice.stMachineConfig.bApplyLabelInPassthrough), bInhibitReset := FALSE, bInternalReset := FALSE, aAlarmsSettings := gMessage.aAlarmsSettings, nAlarmIndex := nAlarmIndex, sMsgInfo := gMessage.stAlarmTable.aMsgHMI[nAlarmIndex], stMsgAux := gMessage.stAlarmTable.aMsgAux[nAlarmIndex]);

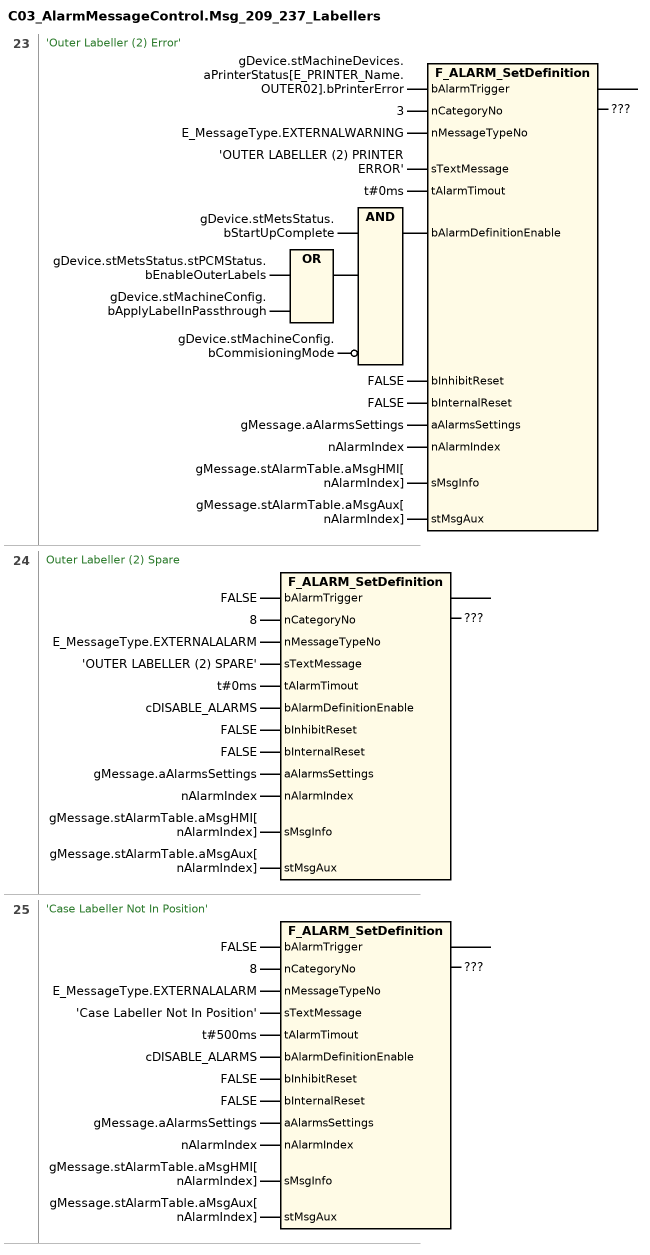
// NETWORK 23
// 'Outer Labeller (2) Error'
F_ALARM_SetDefinition(bAlarmTrigger := gDevice.stMachineDevices.aPrinterStatus[E_PRINTER_Name.OUTER02].bPrinterError, nCategoryNo := 3, nMessageTypeNo := E_MessageType.EXTERNALWARNING, sTextMessage := 'OUTER LABELLER (2) PRINTER ERROR', tAlarmTimout := t#0ms, bAlarmDefinitionEnable := gDevice.stMetsStatus.bStartUpComplete AND (gDevice.stMetsStatus.stPCMStatus.bEnableOuterLabels OR gDevice.stMachineConfig.bApplyLabelInPassthrough) AND NOT gDevice.stMachineConfig.bCommisioningMode, bInhibitReset := FALSE, bInternalReset := FALSE, aAlarmsSettings := gMessage.aAlarmsSettings, nAlarmIndex := nAlarmIndex, sMsgInfo := gMessage.stAlarmTable.aMsgHMI[nAlarmIndex], stMsgAux := gMessage.stAlarmTable.aMsgAux[nAlarmIndex]);

// NETWORK 24
// Outer Labeller (2) Spare
F_ALARM_SetDefinition(bAlarmTrigger := FALSE, nCategoryNo := 8, nMessageTypeNo := E_MessageType.EXTERNALALARM, sTextMessage := 'OUTER LABELLER (2) SPARE', tAlarmTimout := t#0ms, bAlarmDefinitionEnable := cDISABLE_ALARMS, bInhibitReset := FALSE, bInternalReset := FALSE, aAlarmsSettings := gMessage.aAlarmsSettings, nAlarmIndex := nAlarmIndex, sMsgInfo := gMessage.stAlarmTable.aMsgHMI[nAlarmIndex], stMsgAux := gMessage.stAlarmTable.aMsgAux[nAlarmIndex]);

// NETWORK 25
// 'Case Labeller Not In Position'
F_ALARM_SetDefinition(bAlarmTrigger := FALSE, nCategoryNo := 8, nMessageTypeNo := E_MessageType.EXTERNALALARM, sTextMessage := 'Case Labeller Not In Position', tAlarmTimout := t#500ms, bAlarmDefinitionEnable := cDISABLE_ALARMS, bInhibitReset := FALSE, bInternalReset := FALSE, aAlarmsSettings := gMessage.aAlarmsSettings, nAlarmIndex := nAlarmIndex, sMsgInfo := gMessage.stAlarmTable.aMsgHMI[nAlarmIndex], stMsgAux := gMessage.stAlarmTable.aMsgAux[nAlarmIndex]);

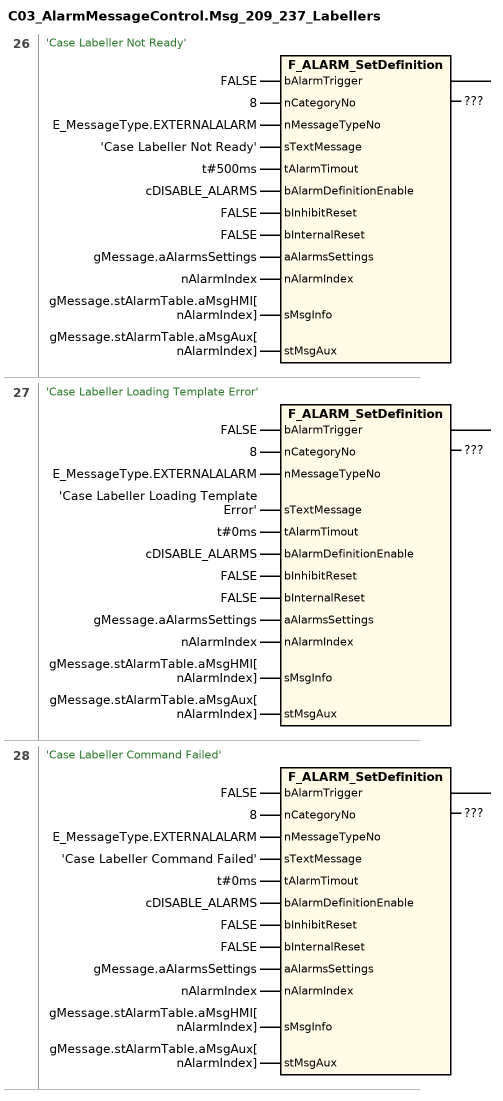
// NETWORK 26
// 'Case Labeller Not Ready'
F_ALARM_SetDefinition(bAlarmTrigger := FALSE, nCategoryNo := 8, nMessageTypeNo := E_MessageType.EXTERNALALARM, sTextMessage := 'Case Labeller Not Ready', tAlarmTimout := t#500ms, bAlarmDefinitionEnable := cDISABLE_ALARMS, bInhibitReset := FALSE, bInternalReset := FALSE, aAlarmsSettings := gMessage.aAlarmsSettings, nAlarmIndex := nAlarmIndex, sMsgInfo := gMessage.stAlarmTable.aMsgHMI[nAlarmIndex], stMsgAux := gMessage.stAlarmTable.aMsgAux[nAlarmIndex]);

// NETWORK 27
// 'Case Labeller Loading Template Error'
F_ALARM_SetDefinition(bAlarmTrigger := FALSE, nCategoryNo := 8, nMessageTypeNo := E_MessageType.EXTERNALALARM, sTextMessage := 'Case Labeller Loading Template Error', tAlarmTimout := t#0ms, bAlarmDefinitionEnable := cDISABLE_ALARMS, bInhibitReset := FALSE, bInternalReset := FALSE, aAlarmsSettings := gMessage.aAlarmsSettings, nAlarmIndex := nAlarmIndex, sMsgInfo := gMessage.stAlarmTable.aMsgHMI[nAlarmIndex], stMsgAux := gMessage.stAlarmTable.aMsgAux[nAlarmIndex]);

// NETWORK 28
// 'Case Labeller Command Failed'
F_ALARM_SetDefinition(bAlarmTrigger := FALSE, nCategoryNo := 8, nMessageTypeNo := E_MessageType.EXTERNALALARM, sTextMessage := 'Case Labeller Command Failed', tAlarmTimout := t#0ms, bAlarmDefinitionEnable := cDISABLE_ALARMS, bInhibitReset := FALSE, bInternalReset := FALSE, aAlarmsSettings := gMessage.aAlarmsSettings, nAlarmIndex := nAlarmIndex, sMsgInfo := gMessage.stAlarmTable.aMsgHMI[nAlarmIndex], stMsgAux := gMessage.stAlarmTable.aMsgAux[nAlarmIndex]);

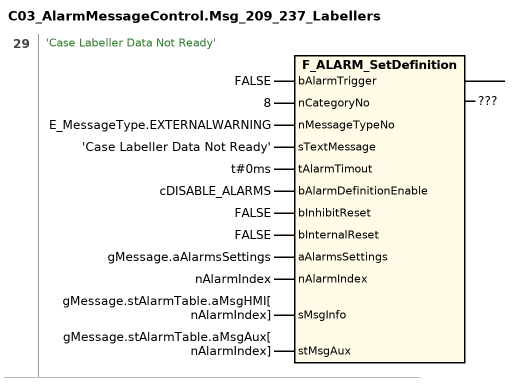
// NETWORK 29
// 'Case Labeller Data Not Ready'
F_ALARM_SetDefinition(bAlarmTrigger := FALSE, nCategoryNo := 8, nMessageTypeNo := E_MessageType.EXTERNALWARNING, sTextMessage := 'Case Labeller Data Not Ready', tAlarmTimout := t#0ms, bAlarmDefinitionEnable := cDISABLE_ALARMS, bInhibitReset := FALSE, bInternalReset := FALSE, aAlarmsSettings := gMessage.aAlarmsSettings, nAlarmIndex := nAlarmIndex, sMsgInfo := gMessage.stAlarmTable.aMsgHMI[nAlarmIndex], stMsgAux := gMessage.stAlarmTable.aMsgAux[nAlarmIndex]);
END_ACTION

ACTION Msg_238_243_Spare:
// note: this text did not pass the execution check against the stored diagram
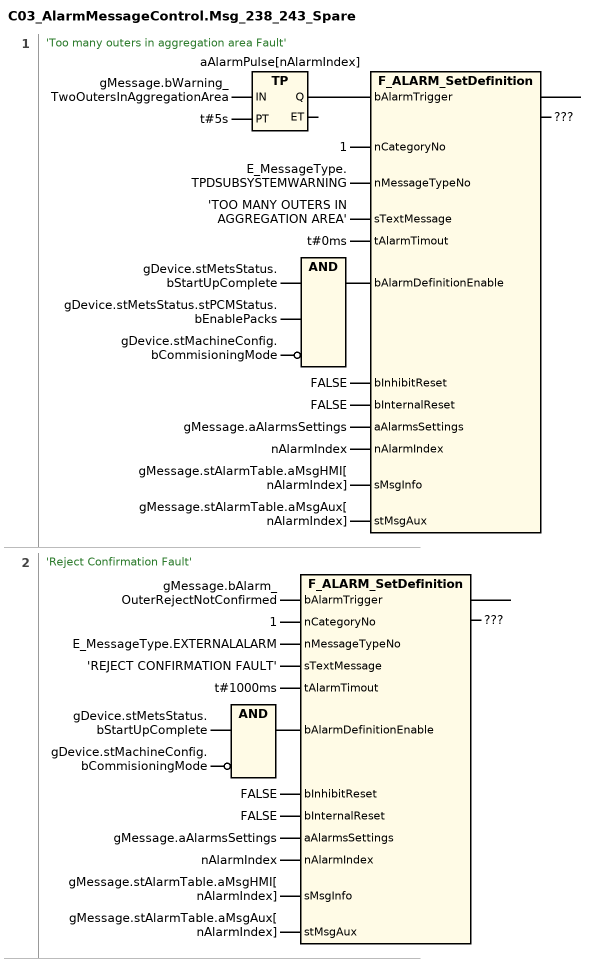
// NETWORK 1
// 'Too many outers in aggregation area Fault'
aAlarmPulse[nAlarmIndex](IN := gMessage.bWarning_TwoOutersInAggregationArea, PT := t#5s); // TP
F_ALARM_SetDefinition(bAlarmTrigger := aAlarmPulse[nAlarmIndex].Q, nCategoryNo := 1, nMessageTypeNo := E_MessageType.TPDSUBSYSTEMWARNING, sTextMessage := 'TOO MANY OUTERS IN AGGREGATION AREA', tAlarmTimout := t#0ms, bAlarmDefinitionEnable := gDevice.stMetsStatus.bStartUpComplete AND gDevice.stMetsStatus.stPCMStatus.bEnablePacks AND NOT gDevice.stMachineConfig.bCommisioningMode, bInhibitReset := FALSE, bInternalReset := FALSE, aAlarmsSettings := gMessage.aAlarmsSettings, nAlarmIndex := nAlarmIndex, sMsgInfo := gMessage.stAlarmTable.aMsgHMI[nAlarmIndex], stMsgAux := gMessage.stAlarmTable.aMsgAux[nAlarmIndex]);

// NETWORK 2
// 'Reject Confirmation Fault'
F_ALARM_SetDefinition(bAlarmTrigger := gMessage.bAlarm_OuterRejectNotConfirmed, nCategoryNo := 1, nMessageTypeNo := E_MessageType.EXTERNALALARM, sTextMessage := 'REJECT CONFIRMATION FAULT', tAlarmTimout := t#1000ms, bAlarmDefinitionEnable := gDevice.stMetsStatus.bStartUpComplete AND NOT gDevice.stMachineConfig.bCommisioningMode, bInhibitReset := FALSE, bInternalReset := FALSE, aAlarmsSettings := gMessage.aAlarmsSettings, nAlarmIndex := nAlarmIndex, sMsgInfo := gMessage.stAlarmTable.aMsgHMI[nAlarmIndex], stMsgAux := gMessage.stAlarmTable.aMsgAux[nAlarmIndex]);

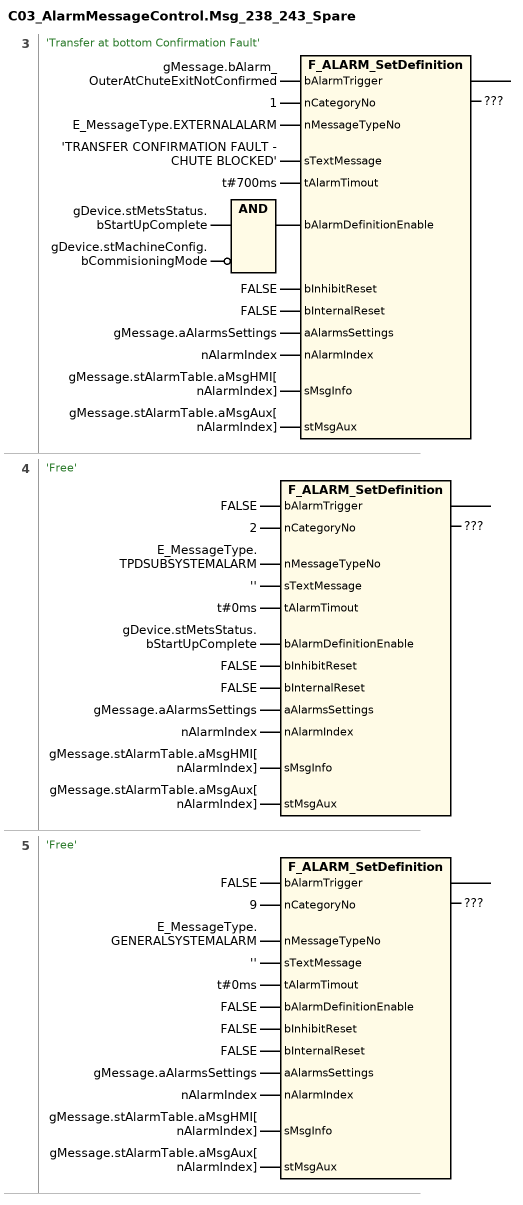
// NETWORK 3
// 'Transfer at bottom Confirmation Fault'
F_ALARM_SetDefinition(bAlarmTrigger := gMessage.bAlarm_OuterAtChuteExitNotConfirmed, nCategoryNo := 1, nMessageTypeNo := E_MessageType.EXTERNALALARM, sTextMessage := 'TRANSFER CONFIRMATION FAULT - CHUTE BLOCKED', tAlarmTimout := t#700ms, bAlarmDefinitionEnable := gDevice.stMetsStatus.bStartUpComplete AND NOT gDevice.stMachineConfig.bCommisioningMode, bInhibitReset := FALSE, bInternalReset := FALSE, aAlarmsSettings := gMessage.aAlarmsSettings, nAlarmIndex := nAlarmIndex, sMsgInfo := gMessage.stAlarmTable.aMsgHMI[nAlarmIndex], stMsgAux := gMessage.stAlarmTable.aMsgAux[nAlarmIndex]);

// NETWORK 4
// 'Free'
F_ALARM_SetDefinition(bAlarmTrigger := FALSE, nCategoryNo := 2, nMessageTypeNo := E_MessageType.TPDSUBSYSTEMALARM, sTextMessage := '', tAlarmTimout := t#0ms, bAlarmDefinitionEnable := gDevice.stMetsStatus.bStartUpComplete, bInhibitReset := FALSE, bInternalReset := FALSE, aAlarmsSettings := gMessage.aAlarmsSettings, nAlarmIndex := nAlarmIndex, sMsgInfo := gMessage.stAlarmTable.aMsgHMI[nAlarmIndex], stMsgAux := gMessage.stAlarmTable.aMsgAux[nAlarmIndex]);

// NETWORK 5
// 'Free'
F_ALARM_SetDefinition(bAlarmTrigger := FALSE, nCategoryNo := 9, nMessageTypeNo := E_MessageType.GENERALSYSTEMALARM, sTextMessage := '', tAlarmTimout := t#0ms, bAlarmDefinitionEnable := FALSE, bInhibitReset := FALSE, bInternalReset := FALSE, aAlarmsSettings := gMessage.aAlarmsSettings, nAlarmIndex := nAlarmIndex, sMsgInfo := gMessage.stAlarmTable.aMsgHMI[nAlarmIndex], stMsgAux := gMessage.stAlarmTable.aMsgAux[nAlarmIndex]);

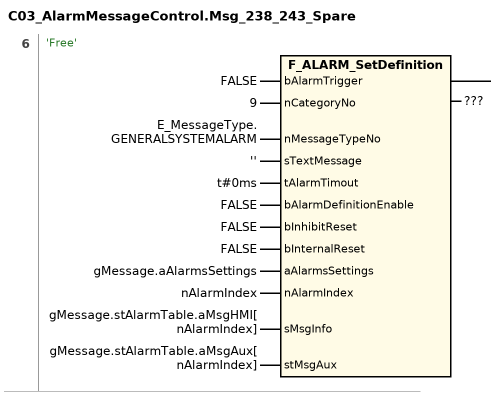
// NETWORK 6
// 'Free'
F_ALARM_SetDefinition(bAlarmTrigger := FALSE, nCategoryNo := 9, nMessageTypeNo := E_MessageType.GENERALSYSTEMALARM, sTextMessage := '', tAlarmTimout := t#0ms, bAlarmDefinitionEnable := FALSE, bInhibitReset := FALSE, bInternalReset := FALSE, aAlarmsSettings := gMessage.aAlarmsSettings, nAlarmIndex := nAlarmIndex, sMsgInfo := gMessage.stAlarmTable.aMsgHMI[nAlarmIndex], stMsgAux := gMessage.stAlarmTable.aMsgAux[nAlarmIndex]);
END_ACTION

ACTION Msg_244_253_DB:
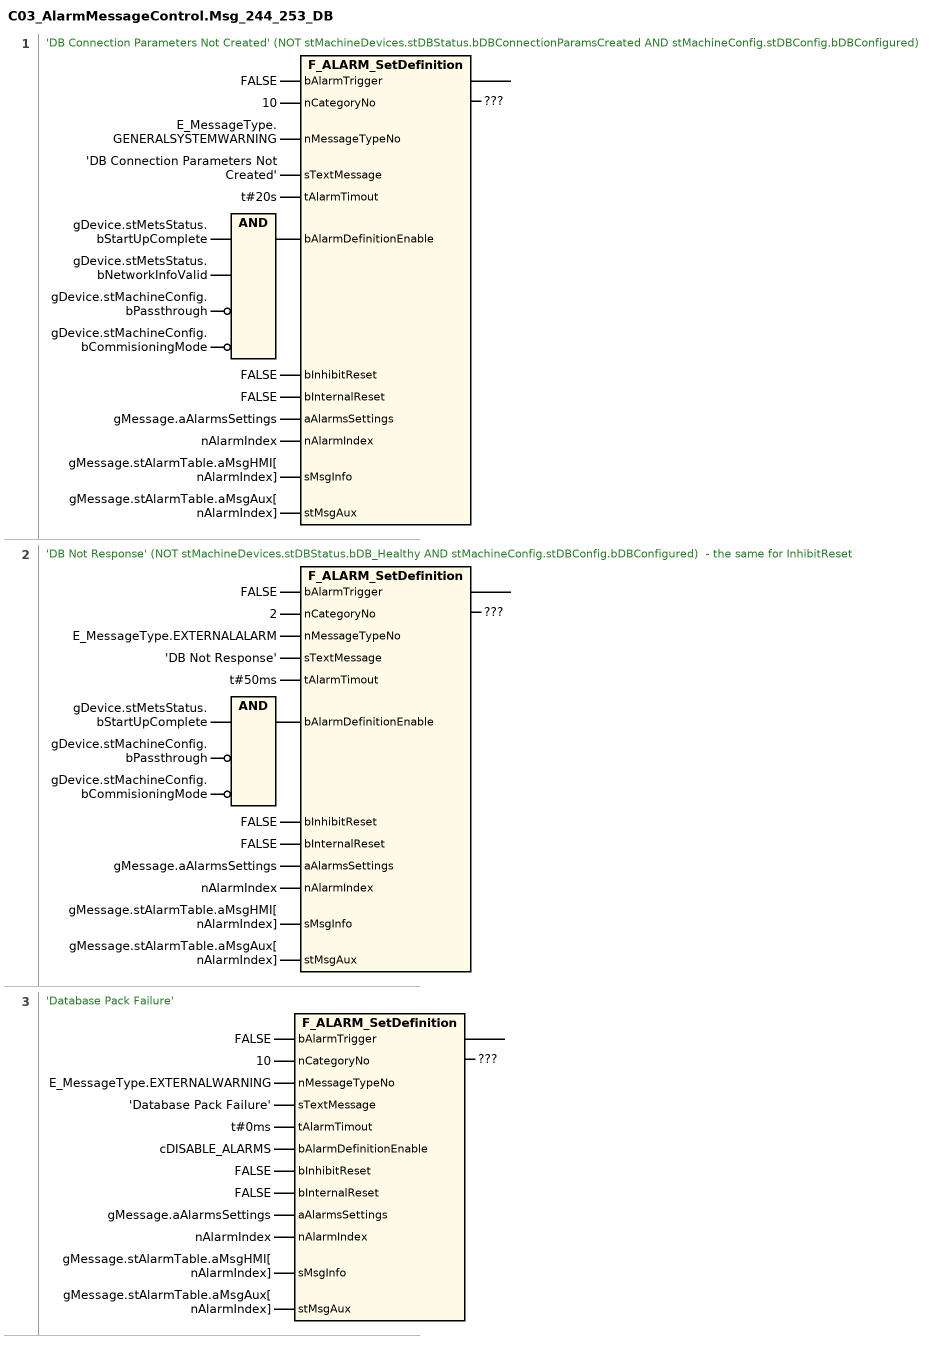
// NETWORK 1
// 'DB Connection Parameters Not Created' (NOT stMachineDevices.stDBStatus.bDBConnectionParamsCreated AND stMachineConfig.stDBConfig.bDBConfigured)
F_ALARM_SetDefinition(bAlarmTrigger := FALSE, nCategoryNo := 10, nMessageTypeNo := E_MessageType.GENERALSYSTEMWARNING, sTextMessage := 'DB Connection Parameters Not Created', tAlarmTimout := t#20s, bAlarmDefinitionEnable := gDevice.stMetsStatus.bStartUpComplete AND gDevice.stMetsStatus.bNetworkInfoValid AND NOT gDevice.stMachineConfig.bPassthrough AND NOT gDevice.stMachineConfig.bCommisioningMode, bInhibitReset := FALSE, bInternalReset := FALSE, aAlarmsSettings := gMessage.aAlarmsSettings, nAlarmIndex := nAlarmIndex, sMsgInfo := gMessage.stAlarmTable.aMsgHMI[nAlarmIndex], stMsgAux := gMessage.stAlarmTable.aMsgAux[nAlarmIndex]);

// NETWORK 2
// 'DB Not Response' (NOT stMachineDevices.stDBStatus.bDB_Healthy AND stMachineConfig.stDBConfig.bDBConfigured)  - the same for InhibitReset
F_ALARM_SetDefinition(bAlarmTrigger := FALSE, nCategoryNo := 2, nMessageTypeNo := E_MessageType.EXTERNALALARM, sTextMessage := 'DB Not Response', tAlarmTimout := t#50ms, bAlarmDefinitionEnable := gDevice.stMetsStatus.bStartUpComplete AND NOT gDevice.stMachineConfig.bPassthrough AND NOT gDevice.stMachineConfig.bCommisioningMode, bInhibitReset := FALSE, bInternalReset := FALSE, aAlarmsSettings := gMessage.aAlarmsSettings, nAlarmIndex := nAlarmIndex, sMsgInfo := gMessage.stAlarmTable.aMsgHMI[nAlarmIndex], stMsgAux := gMessage.stAlarmTable.aMsgAux[nAlarmIndex]);

// NETWORK 3
// 'Database Pack Failure'
F_ALARM_SetDefinition(bAlarmTrigger := FALSE, nCategoryNo := 10, nMessageTypeNo := E_MessageType.EXTERNALWARNING, sTextMessage := 'Database Pack Failure', tAlarmTimout := t#0ms, bAlarmDefinitionEnable := cDISABLE_ALARMS, bInhibitReset := FALSE, bInternalReset := FALSE, aAlarmsSettings := gMessage.aAlarmsSettings, nAlarmIndex := nAlarmIndex, sMsgInfo := gMessage.stAlarmTable.aMsgHMI[nAlarmIndex], stMsgAux := gMessage.stAlarmTable.aMsgAux[nAlarmIndex]);

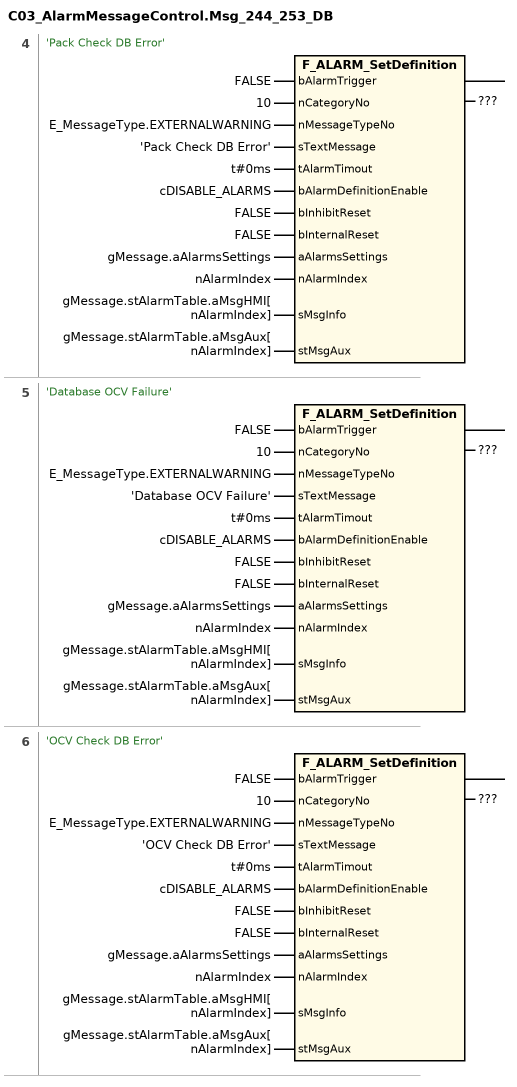
// NETWORK 4
// 'Pack Check DB Error'
F_ALARM_SetDefinition(bAlarmTrigger := FALSE, nCategoryNo := 10, nMessageTypeNo := E_MessageType.EXTERNALWARNING, sTextMessage := 'Pack Check DB Error', tAlarmTimout := t#0ms, bAlarmDefinitionEnable := cDISABLE_ALARMS, bInhibitReset := FALSE, bInternalReset := FALSE, aAlarmsSettings := gMessage.aAlarmsSettings, nAlarmIndex := nAlarmIndex, sMsgInfo := gMessage.stAlarmTable.aMsgHMI[nAlarmIndex], stMsgAux := gMessage.stAlarmTable.aMsgAux[nAlarmIndex]);

// NETWORK 5
// 'Database OCV Failure'
F_ALARM_SetDefinition(bAlarmTrigger := FALSE, nCategoryNo := 10, nMessageTypeNo := E_MessageType.EXTERNALWARNING, sTextMessage := 'Database OCV Failure', tAlarmTimout := t#0ms, bAlarmDefinitionEnable := cDISABLE_ALARMS, bInhibitReset := FALSE, bInternalReset := FALSE, aAlarmsSettings := gMessage.aAlarmsSettings, nAlarmIndex := nAlarmIndex, sMsgInfo := gMessage.stAlarmTable.aMsgHMI[nAlarmIndex], stMsgAux := gMessage.stAlarmTable.aMsgAux[nAlarmIndex]);

// NETWORK 6
// 'OCV Check DB Error'
F_ALARM_SetDefinition(bAlarmTrigger := FALSE, nCategoryNo := 10, nMessageTypeNo := E_MessageType.EXTERNALWARNING, sTextMessage := 'OCV Check DB Error', tAlarmTimout := t#0ms, bAlarmDefinitionEnable := cDISABLE_ALARMS, bInhibitReset := FALSE, bInternalReset := FALSE, aAlarmsSettings := gMessage.aAlarmsSettings, nAlarmIndex := nAlarmIndex, sMsgInfo := gMessage.stAlarmTable.aMsgHMI[nAlarmIndex], stMsgAux := gMessage.stAlarmTable.aMsgAux[nAlarmIndex]);

